Fanuc KAREL source: kf00027.KL

-- PROVISIONAL review KL for V770-1; original PC SHA256 8c0a6b76168a3bf9ccd88c4e13a8bf2134e8c917aeac61a8fbc807b50ba6b280
-- Incomplete behavior may be omitted. Consult companion uncertainty JSON. Do not deploy.
PROGRAM KF00027
%NOLOCKGROUP
VAR
  I : INTEGER
  J : INTEGER
  X : REAL
  Y : REAL
  B : BOOLEAN
  C : BOOLEAN
  TXT : STRING[80]
  TXT2 : STRING[80]
  STATUS : INTEGER
-- UNRESOLVED_DECL AI type=002010
-- UNRESOLVED_DECL BI type=002010
-- UNRESOLVED_DECL P type=000102
-- UNRESOLVED_DECL JP type=000199
-- UNRESOLVED_DECL PF type=000101
-- UNRESOLVED_DECL V1 type=000013
-- UNRESOLVED_DECL V2 type=000013
BEGIN
  -- UNRESOLVED_PC offsets 5-16; opcodes 3F,75
  -- UNRESOLVED_PC offsets 21-32; opcodes 3F,75
  -- UNRESOLVED_PC offsets 37-56; opcodes 73,73,85,23
  -- UNRESOLVED_PC offsets 61-65; opcodes 7F
END KF00027
